INTERFACE I_PackML_ExternalController

PROPERTY Control : I_PackML_Control
SET
END_SET
END_PROPERTY

METHOD ModeChanged
VAR_INPUT
    NewMode : E_PMLUnitMode;
END_VAR
END_METHOD

METHOD StateChanged
VAR_INPUT
    NewState : E_PMLCommand;
END_VAR
END_METHOD

END_INTERFACE

(* stored: Version 1.1.0.1, ProductVersion 3.1.4024.12
   Itf I_PackML_ExternalController: Id {7432f408-274f-47ce-b8be-362011fb55e5}
   Property Control: Id {771f3b04-91f5-43a8-8f54-e3fe4eda6c87}
   Set Set: Id {45c6b3b0-6b70-49d7-859c-643dc741120d}
   Method ModeChanged: Id {3ac5a7bd-15d2-4d47-8be6-44d74412d718}
   Method StateChanged: Id {c930b1eb-e910-48fb-9de7-42aa1a5f7aa8} *)
